FUNCTION_BLOCK Turntable
VAR_INPUT



END_VAR
VAR_OUTPUT

	bTurn 		: BOOL;
	bRollPlus	: BOOL;
	bRollMinus 	: BOOL;
	bFrontLimit : BOOL;
	bBackLimit	: BOOL;
	
END_VAR
VAR

	fbFrontLimit : Sensor;
	fbBackLimit : Sensor;
	
	fbTurn : BoolOut;
	fbRollPlus : BoolOut;
	fbRollMinus : BoolOut;
	
END_VAR

fbFrontLimit();
fbBackLimit();

bTurn := fbTurn.getValue;
bRollPlus := fbRollPlus.getValue;
bRollMinus := fbRollMinus.getValue;
bFrontLimit := fbFrontLimit.bSignal;
bBackLimit	:= fbBackLimit.bSignal;

METHOD RollMinus : BOOL
VAR_INPUT
END_VAR
fbRollMinus.setValue := TRUE;
fbRollPlus.setValue := FALSE;
END_METHOD

METHOD RollPlus : BOOL
VAR_INPUT
END_VAR
fbRollPlus.setValue := TRUE;
fbRollMinus.setValue := FALSE;
END_METHOD

METHOD StopRolling : BOOL
VAR_INPUT
END_VAR
fbRollMinus.setValue := FALSE;
fbRollPlus.setValue := FALSE;
END_METHOD

METHOD Turn : BOOL
VAR_INPUT
END_VAR
fbTurn.setValue := TRUE;
END_METHOD

METHOD Unturn : BOOL
VAR_INPUT
END_VAR
fbTurn.setValue := FALSE;
END_METHOD

END_FUNCTION_BLOCK

(* stored: Version 1.1.0.1, ProductVersion 3.1.4024.2
   POU Turntable: Id {5a7b578a-85d4-41c6-b84c-ca292559fdbd}, SpecialFunc None
   Method RollMinus: Id {207a62c8-6d7f-4007-bdf2-cf32530a58e7}
   Method RollPlus: Id {ec53d457-a63c-4bd8-a2a4-20f5059e9164}
   Method StopRolling: Id {2419d82f-e24f-4160-8b39-e47e4f6a13da}
   Method Turn: Id {1c28c895-9ab6-4303-bd55-9592fe01ec59}
   Method Unturn: Id {b36ebc82-ea4b-4c3f-b5ca-518e79da2d00} *)
